// TIA Portal V20 export
// export: Created 2025-12-01T14:56:09.9677032Z, ExportSetting None, DisplayName Totally Integrated Automation Portal, DisplayVersion V20 Update 3, DisplayName TIA Portal Openness, DisplayVersion V20 Update 3, DisplayName TIA Portal Version Control Interface, DisplayVersion V20 Update 3, DisplayName STEP 7 Professional, DisplayVersion V20 Update 3, DisplayName STEP 7 Safety, DisplayVersion V20 Update 2, DisplayName WinCC Basic/Comfort/Advanced, DisplayVersion V20 Update 3, DisplayName WinCC Professional, DisplayVersion V20 Update 3, DisplayName WinCC Unified, DisplayVersion V20 Update 3
TYPE "LPNDR_typeMrpInformation"
   STRUCT
      mrpRole : UInt;   // 0=disabled, 1=client, 2=manager, 3=manager(auto)
      domainName : String[240];
   END_STRUCT;
END_TYPE
